% RSLogix 500 project Intro to PLC Job HO4 Adam Huels.RSS, saved by version 10.00.00.00 %
PROJECT "UNTITLED"    % processor: Bul.1763 MicroLogix 1100 Series B %

PROGRAM FILES
  LAD 2   8 rungs

DATA FILES
  O0 OUTPUT  4 elements
  I1 INPUT  6 elements
  S2 STATUS  66 elements
  B3 BINARY  1 elements
  T4 TIMER  1 elements
  C5 COUNTER  1 elements
  R6 CONTROL  1 elements
  N7 INTEGER  1 elements
  F8 FLOAT  1 elements

LADDER 2
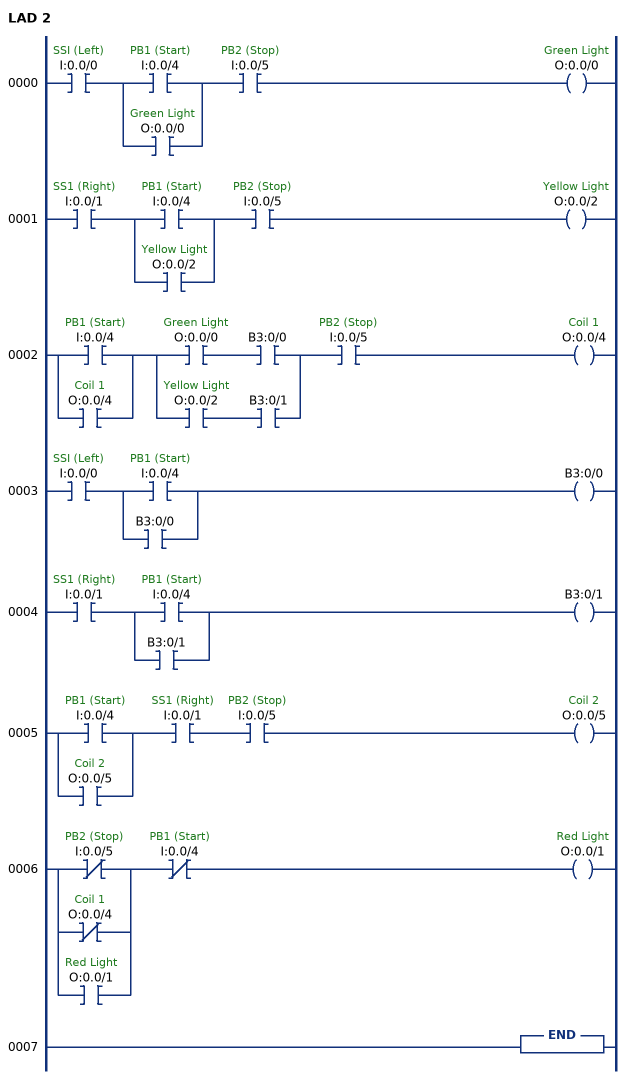
% Rung: 0 %
SOR XIC I:0.0/0 BST XIC I:0.0/4 NXB XIC O:0.0/0 BND XIC I:0.0/5 OTE O:0.0/0 EOR
%   I:0.0/0  "SSI (Left)" %
%   I:0.0/4  "PB1 (Start)" %
%   O:0.0/0  "Green Light" %
%   I:0.0/5  "PB2 (Stop)" %
% Rung: 1 %
SOR XIC I:0.0/1 BST XIC I:0.0/4 NXB XIC O:0.0/2 BND XIC I:0.0/5 OTE O:0.0/2 EOR
%   I:0.0/1  "SS1 (Right)" %
%   I:0.0/4  "PB1 (Start)" %
%   O:0.0/2  "Yellow Light" %
%   I:0.0/5  "PB2 (Stop)" %
% Rung: 2 %
SOR BST XIC I:0.0/4 NXB XIC O:0.0/4 BND BST XIC O:0.0/0 XIC B3:0/0 NXB XIC O:0.0/2 XIC B3:0/1 BND XIC I:0.0/5 OTE O:0.0/4 EOR
%   I:0.0/4  "PB1 (Start)" %
%   O:0.0/4  "Coil 1" %
%   O:0.0/0  "Green Light" %
%   O:0.0/2  "Yellow Light" %
%   I:0.0/5  "PB2 (Stop)" %
% Rung: 3 %
SOR XIC I:0.0/0 BST XIC I:0.0/4 NXB XIC B3:0/0 BND OTE B3:0/0 EOR
%   I:0.0/0  "SSI (Left)" %
%   I:0.0/4  "PB1 (Start)" %
% Rung: 4 %
SOR XIC I:0.0/1 BST XIC I:0.0/4 NXB XIC B3:0/1 BND OTE B3:0/1 EOR
%   I:0.0/1  "SS1 (Right)" %
%   I:0.0/4  "PB1 (Start)" %
% Rung: 5 %
SOR BST XIC I:0.0/4 NXB XIC O:0.0/5 BND XIC I:0.0/1 XIC I:0.0/5 OTE O:0.0/5 EOR
%   I:0.0/4  "PB1 (Start)" %
%   O:0.0/5  "Coil 2" %
%   I:0.0/1  "SS1 (Right)" %
%   I:0.0/5  "PB2 (Stop)" %
% Rung: 6 %
SOR BST XIO I:0.0/5 NXB XIO O:0.0/4 NXB XIC O:0.0/1 BND XIO I:0.0/4 OTE O:0.0/1 EOR
%   I:0.0/5  "PB2 (Stop)" %
%   O:0.0/4  "Coil 1" %
%   O:0.0/1  "Red Light" %
%   I:0.0/4  "PB1 (Start)" %
% Rung: 7 %
SOR END EOR
